FUNCTION_BLOCK Fixture
  (* Version 1.0, 2007-08-23, Goran Cengic, Chalmers *)
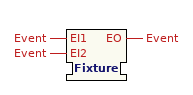
  EVENT_INPUT
    EI1;
    EI2;
  END_EVENT
  EVENT_OUTPUT
    EO;
  END_EVENT
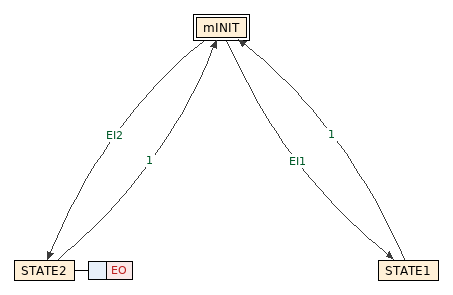
  EC_STATES
    mINIT;
    STATE1;
    STATE2 : -> EO;
  END_STATES
  EC_TRANSITIONS
    mINIT TO STATE1 := EI1;
    STATE1 TO mINIT := 1;
    mINIT TO STATE2 := EI2;
    STATE2 TO mINIT := 1;
  END_TRANSITIONS
END_FUNCTION_BLOCK
(* other elements stored in the file *)
(* ECAction Algorithm="OpenClamp" / *)
(* ECAction Algorithm="PushOut" Output="EO"/ *)
(* Algorithm Name="OpenClamp"> <Other Language="Java" Text="System.out.println(&#34;Opening Clamp!&#34;);" /> </Algorithm> <Algorithm Name="PushOut"> <Other Language="Java" Text="System.out.println(&#34;Pushing Out!&#34;);" /> </Algorithm *)
